// TIA Portal project "Soru2" (V15)

(* hardware
DEVICE "S7-1200 station_1"  S7-1200 Station
   slot 0: "Rack_0"  S7-1200 Rack  Rack  V1.0
   slot 1: "PLC_1"  CPU 1214C DC/DC/DC  6ES7 214-1AG40-0XB0  V4.2
*)

// ===== PLC "PLC_1"  CPU 1214C DC/DC/DC =====

VAR_GLOBAL   // PLC tag table "Default tag table"
   "durdru" AT %I0.0 : Bool;
   "basla" AT %I0.1 : Bool;
   "Motor_1" AT %Q0.0 : Bool;
   "Motor_2" AT %Q0.1 : Bool;
   "Motor_3" AT %Q0.2 : Bool;
END_VAR

// folder: System blocks/Program resources

DATA_BLOCK "zman1"   // DB1
{ S7_Optimized_Access := 'TRUE' }
AUTHOR : Simatic
FAMILY : IEC
NAME : IEC_TMR
VERSION : 1.0
// stored: InstanceOfName IEC_TIMER
"IEC_TIMER"
BEGIN
END_DATA_BLOCK

DATA_BLOCK "zman2"   // DB2
{ S7_Optimized_Access := 'TRUE' }
AUTHOR : Simatic
FAMILY : IEC
NAME : IEC_TMR
VERSION : 1.0
// stored: InstanceOfName IEC_TIMER
"IEC_TIMER"
BEGIN
END_DATA_BLOCK

DATA_BLOCK "zman3"   // DB3
{ S7_Optimized_Access := 'TRUE' }
AUTHOR : Simatic
FAMILY : IEC
NAME : IEC_TMR
VERSION : 1.0
// stored: InstanceOfName IEC_TIMER
"IEC_TIMER"
BEGIN
END_DATA_BLOCK

// folder: (top level)

ORGANIZATION_BLOCK "Main"   // OB1, LAD, ProgramCycle
TITLE = "Main Program Sweep (Cycle)"
{ S7_Optimized_Access := 'TRUE' }
VERSION : 0.1
   VAR_INPUT
      Initial_Call : Bool;   // Initial call of this OB
      Remanence : Bool;   // =True, if remanent data are available
   END_VAR
BEGIN

REGION Network 1
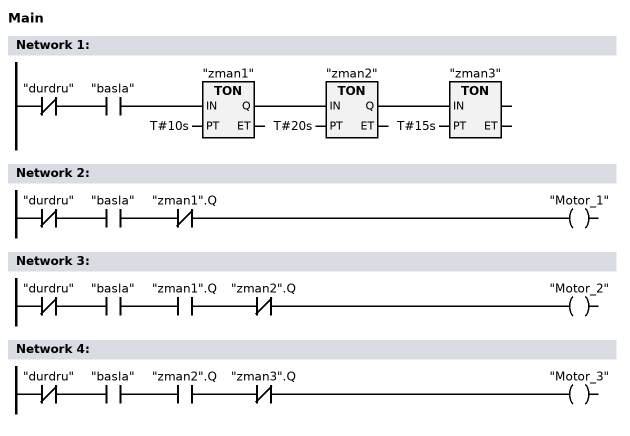
   "zman1".TON(IN := NOT "durdru" AND "basla", PT := T#10s);
   "zman2".TON(IN := "zman1".Q, PT := T#20s);
   "zman3".TON(IN := "zman2".Q, PT := T#15s);
END_REGION

REGION Network 2
   RUNG wire#powerrail
      I_Contact( "durdru" )
      Contact( "basla" )
      I_Contact( "zman1".Q )
      Coil( "Motor_1" )
   END_RUNG
   // the same network as SCL:
   "Motor_1" := NOT "durdru" AND "basla" AND NOT "zman1".Q;
END_REGION

REGION Network 3
   RUNG wire#powerrail
      I_Contact( "durdru" )
      Contact( "basla" )
      Contact( "zman1".Q )
      I_Contact( "zman2".Q )
      Coil( "Motor_2" )
   END_RUNG
   // the same network as SCL:
   "Motor_2" := NOT "durdru" AND "basla" AND "zman1".Q AND NOT "zman2".Q;
END_REGION

REGION Network 4
   RUNG wire#powerrail
      I_Contact( "durdru" )
      Contact( "basla" )
      Contact( "zman2".Q )
      I_Contact( "zman3".Q )
      Coil( "Motor_3" )
   END_RUNG
   // the same network as SCL:
   "Motor_3" := NOT "durdru" AND "basla" AND "zman2".Q AND NOT "zman3".Q;
END_REGION
END_ORGANIZATION_BLOCK